(*
Enables pairing with receivers and emitting, but not casting to `I_Component`.
*)
INTERFACE I_SignalEmit

(*
Emits an argument through the signal's broadcasting system.  
If no argument is provided, it defaults to emitting the associated tag.
Returns:
- `Ok` - On Success
- `Err.InfLoop` - Upon recursive call attempt
*)
METHOD Emit : Result
VAR_INPUT
	iArg			: I_Arg := 0;
END_VAR
END_METHOD

(*
Emits an argument to a specified receiver.
Returns:
- `Ok` - If the emission is successful.
- `Err.Itf0` - If the receiver interface is invalid.
- `Err.InfLoop` - Upon recursive call attempt
*)
METHOD EmitTo : Result
VAR_INPUT
	iReceiver		: I_Receiver;
	iArg			: I_Arg := 0;
END_VAR
END_METHOD

(*
Sets an Tag.Option property of an internal Tag. Chainable.
*)
METHOD Option : REFERENCE TO Signal
VAR_INPUT
	sOption		: Str;
END_VAR
END_METHOD

(*
Pairs the signal with a receiver.  
Returns:
- `Ok` - If pairing is successful.
- `Err.Itf0` - If the receiver interface is invalid.
- `Err.IncArg` - If the `I_Receiver` is invalid.
- `Err.ItfEq` - If the `I_Receiver` is already paired with this `I_Signal`.
- `Err.Ovf` - If there is no space for another pairing.
*)
METHOD Pair : Result
VAR_INPUT
	iReceiver		: I_Receiver;
END_VAR
END_METHOD

(*
Provides access to the tag associated with the signal.
*)
PROPERTY Tag : I_Tag
GET
END_GET
END_PROPERTY

(*
Unpairs the signal from a specified receiver.
Returns:
- `Ok` - If unpairing is successful.
- `Err.Itf0` - If the receiver interface is invalid.
- `Err.IncArg` - If the `I_Receiver` is invalid.
- `Err.NoMatch` - If `I_Signal` is not paired with this `I_Receiver`.
*)
METHOD Unpair : Result
VAR_INPUT
	iReceiver		: I_Receiver;
END_VAR
END_METHOD

END_INTERFACE

(* stored: Version 1.1.0.1
   Itf I_SignalEmit: Id {609e01a1-b6ea-4fea-abd9-80ec28843d94}
   Method Emit: Id {92a7c3da-021c-46a2-9cd8-62f5dba6bf6c}
   Method EmitTo: Id {76b81514-dc0e-4ebc-aa38-74fb287e595a}
   Method Option: Id {0f6d914b-8b06-423c-b5b9-166095e390b3}
   Method Pair: Id {84e28503-3123-4a24-91ee-88e64b2e187b}
   Property Tag: Id {3075fdb7-eb8c-4274-95ea-6ec5a2600afc}
   Get Get: Id {83c96f7e-bf2d-42c3-ab5d-b460d6ba2728}
   Method Unpair: Id {e8a625b4-f16a-4019-9c13-4f5291029ddb} *)
